Staubli VAL3: ArcLength.pgx

public program ArcLength(trsf x_trFirst, trsf x_trCenter, trsf x_trEnd, num& x_nLength)
  local trsf l_trTrsf[3]
  local bool l_bBool
begin


  //获得圆弧长度
  //如果报错,那么就返回值为0


  x_nLength=0

  l_trTrsf[0]=x_trFirst
  l_trTrsf[1]=x_trCenter
  l_trTrsf[2]=x_trEnd

  call GetArcLength(l_trTrsf,x_nLength,l_bBool)
  if !l_bBool
    x_nLength=0
  endIf



end
